FUNCTION_BLOCK ChangeDetectComp (* Composite Function Block Type *)
  (* Standard: 61499-2 *)
  (* Version 0.0, 7/13/2023, Cheyan, Schneider Electric, template *)
  PACKAGE Main;
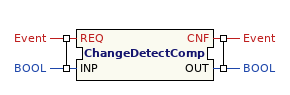
  EVENT_INPUT
    REQ WITH INP; (* Normal Execution Request *)
  END_EVENT
  EVENT_OUTPUT
    CNF WITH OUT; (* Execution Confirmation *)
  END_EVENT
  VAR_INPUT
    INP : BOOL; (* Input event qualifier *)
  END_VAR
  VAR_OUTPUT
    OUT : BOOL; (* Output event qualifier *)
  END_VAR
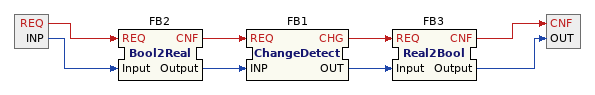
  FBS
    FB1 : ChangeDetect;
    FB2 : Bool2Real;
    FB3 : Real2Bool;
  END_FBS
  EVENT_CONNECTIONS
    FB2.CNF TO FB1.REQ;
    REQ TO FB2.REQ;
    FB1.CHG TO FB3.REQ;
    FB3.CNF TO CNF;
  END_CONNECTIONS
  DATA_CONNECTIONS
    FB2.Output TO FB1.INP;
    INP TO FB2.Input;
    FB1.OUT TO FB3.Input;
    FB3.Output TO OUT;
  END_CONNECTIONS
END_FUNCTION_BLOCK
